PROGRAM MAIN
VAR
	// Define the top level Machine as defined in the Application/01_MachineModules folder here
	fbMyMachine				: FB_TestMachine;	
	fbMainHMIConnection		: FB_MainHMI_Connection;

	bInitialized			: BOOL;
END_VAR

CyclicLogic();

METHOD CyclicLogic : BOOL
VAR_INPUT
END_VAR
IF NOT bInitialized THEN
	Initialize();
	bInitialized := TRUE;
END_IF

//The Top level machine CyclicLogic call should be made here, all sub modules should be called from within their respective parent CyclicLogic methods
fbMyMachine.CyclicLogic();


// Add other Main CyclicLogic here
fbMainHMIConnection();
//test
END_METHOD

METHOD Initialize : BOOL
VAR_INPUT
END_VAR
//Top level machine initialization should happen here, in the main initialization method. Each subsequent "layer" of modules will be named within their respective "parent" intialize method
fbMainHMIConnection.sTopLevelMachine := fbMyMachine.ModuleName;

fbMyMachine.MasterDataStructure_Adder  	:= fbMainHMIConnection.DataStructure_Adder;
fbMyMachine.Enabled 					:=  TRUE;
fbMyMachine.ModuleName 					:=  'Test Machine';
fbMyMachine.ModuleID 					:=  1;
fbMyMachine.AncestorIDs 				:= '';

fbMainHMIConnection(sTopLevelMachine 	:= fbMyMachine.ModuleName);
END_METHOD

END_PROGRAM

(* stored: Version 1.1.0.1, ProductVersion 3.1.4024.9
   POU MAIN: Id {ea287bb8-b345-4656-b603-ee461cbe7d52}, SpecialFunc None
   Method CyclicLogic: Id {5d3afc59-d698-49af-9648-a60196d60bb0}
   Method Initialize: Id {0c84ac41-2efe-4430-b0e8-a78a2e3a34ca} *)
